TYPE ST_INTERCEPTOR :
STRUCT
	check:	BOOL;
	desc:	T_SHORT_STR;
END_STRUCT
END_TYPE

(* stored: Version 1.1.0.1, ProductVersion 3.1.4026.18
   DUT ST_INTERCEPTOR: Id {2b4d557f-cdec-4aa4-9bf1-c67a1ac49246} *)
